// TwinCAT 3 PLC project PLC
// Title: abc
// Company: abc
// ProjectVersion: 1.0
// ProgramVersion: 3.1.0.8
// libraries:
//   Tc2_Standard, * (Beckhoff Automation GmbH)
//   Tc2_System, * (Beckhoff Automation GmbH)
//   Tc3_Interfaces, * (Beckhoff Automation GmbH)
//   Tc3_Module, * (Beckhoff Automation GmbH)
// project tree:
//   DUTs/ MyComplexStruct.TcDUT, MYSTRUCT.TcDUT, PLCStruct.TcDUT (not stored), TComplexStruct.TcDUT (not stored), TSimpleStruct.TcDUT
//   GVLs/ GVL.TcGVL (not stored)
//   / PlcTask.TcTTO
//   POUs/ FB_Math.TcPOU (not stored), MAIN.TcPOU
//   Version/ Global_Version.TcGVL (not stored)
// real-time tasks:
//   TASK PlcTask: cycle T#10ms, priority 20, ADS port 350

CONFIGURATION PLC
    RESOURCE PLC ON TwinCAT3
        TASK PlcTask(INTERVAL := T#10ms, PRIORITY := 20);
        PROGRAM MAIN WITH PlcTask : MAIN;
    END_RESOURCE
END_CONFIGURATION

// ---- DUTs/MyComplexStruct.TcDUT
{attribute 'pack_mode' := '1'} 
TYPE MyComplexStruct :
STRUCT
	a : BOOL;
	b : INT;
	c : DINT;
	d : MYSTRUCT;
END_STRUCT
END_TYPE

// ---- DUTs/MYSTRUCT.TcDUT
{attribute 'pack_mode' := '1'} 
TYPE MYSTRUCT :
STRUCT
	a : BOOL;
	b : INT;
	c : DINT;
END_STRUCT
END_TYPE

// ---- DUTs/TSimpleStruct.TcDUT
TYPE TSimpleStruct :
STRUCT
	lrealVal: 	LREAL  	:= 1.23;
	dintVal1:	DINT 	 := 120000;
END_STRUCT
END_TYPE

// ---- POUs/MAIN.TcPOU
PROGRAM MAIN
VAR
	//Sample 01 and 02
	nCounter     AT %MD0 :DWORD;
	TP_1		: TP;
	TOGGEL		: BOOL;

	//Sample03
	 boolVal   : BOOL;
	 intVal    : INT;
	 dintVal   : DINT;
	 sintVal   : SINT;
	 lrealVal  : LREAL;
	 realVal   : REAL;
	 stringVal : STRING(20);
	 
	 myComplexStruct : MyComplexStruct;
	 
	//Sample10
	text : STRING[30] := 'Hello TwinCAT';
	
	//Sample11
	Time1:TIME := T#21H33M23S231MS;
    Date1:DT:=DT#1993-06-12-15:36:55.40;
	
	//Sample12
	PLCArray : ARRAY [0..99] OF INT;
  	Index: BYTE;
	
	//Sample13
	PLCStruct : PLCStruct;	
	
	//Sample14
	(*primitive Types*)
	bool1:BOOL := FALSE;
	int1:INT := 30000;
	dint1:DINT:=125000;
	usint1:USINT:=200;
	real1:REAL:= 1.2;
	lreal1:LREAL:=3.5;

	(*string Types*)
	str1:STRING := 'this is a test string';
	str2:STRING(5) := 'hallo';

	(*struct Types*)
	complexStruct1 : TComplexStruct;
	
	//Sample22
	uintValue 	: UDINT 	:= 54321;
	boolValue	: BOOL 		:= TRUE;
	dintValue	: DINT		:= -12345678;
	
	//Sample30
	fbMath	: FB_MATH;
	TON1: TON;
END_VAR



//Sample 01 and 02
nCounter := nCounter + 1;

//Sample 03
sintVal := sintVal + 1;
dintVal := dintVal + 5;
realVal := realVal + 0.1;
lrealVal := lrealVal + 0.1;

boolVal := FALSE;
TON1(IN:= TRUE, PT:= T#200MS, Q=> boolVal);
IF boolVal THEN
	IF intval > 12 THEN
		intval := 0;
	END_IF
	intVal := intVal + 1;
	stringVal := LEFT(Text, intVal);
	TON1(IN:= FALSE);
END_IF

//Sample12
FOR Index := 0 TO 99 DO
  PLCArray[Index] := 3500 + INDEX;
END_FOR

myComplexStruct.a := true;

END_PROGRAM
